Yaskawa INFORM job: SKRZYNIA_5040_90_STOPNI_20BR.JBI

/JOB
//NAME SKRZYNIA_5040_90_STOPNI_20BR
///FOLDERNAME 02-SKRZYNIE_JOBS
//POS
///NPOS 545,545,0,38,0,0
///TOOL 0
///POSTYPE PULSE
///PULSE
C00000=0,-52280,40443,0,6876,0
C00001=82314,-24956,17040,59626,-27382,6248
C00002=93910,-8625,17040,59626,-43355,6248
C00003=98846,-1061,-42166,80308,-57081,-16120
C00004=100452,6057,-48127,85711,-56704,-21322
C00005=95573,33077,-33257,84645,-64023,-26851
C00006=94102,33899,-31937,85246,-63371,-26689
C00007=95573,33077,-33257,84645,-64023,-26851
C00008=94862,31071,-36438,85313,-63677,-27192
C00009=95573,33077,-33257,84645,-64023,-26851
C00010=95263,33142,-33256,84677,-63995,-26850
C00011=95263,33142,-33256,84677,-63995,-26850
C00012=94017,33843,-32133,85187,-63445,-26710
C00013=95263,33142,-33256,84677,-63995,-26850
C00014=94657,31439,-35966,85248,-63701,-27141
C00015=95263,33142,-33256,84677,-63995,-26850
C00016=95260,33144,-33256,84678,-63995,-26850
C00017=95260,33144,-33256,84678,-63995,-26850
C00018=94022,33838,-32141,85183,-63448,-26711
C00019=95260,33144,-33256,84678,-63995,-26850
C00020=94618,31343,-36117,85281,-63684,-27157
C00021=95260,33144,-33256,84678,-63995,-26850
C00022=95258,25631,32269,66559,-75499,-2416
C00023=95258,25631,32269,66559,-75499,-2416
C00024=94181,26497,33533,66410,-74896,-2191
C00025=95658,30184,39035,66708,-78559,-2356
C00026=95217,30377,39331,66881,-79841,-2558
C00027=95258,25631,32269,66559,-75499,-2416
C00028=98811,21047,-15512,99242,-81394,-20987
C00029=98811,21047,-15512,99242,-81394,-20987
C00030=97775,21639,-14693,99563,-80753,-20993
C00031=98811,21047,-15512,99242,-81394,-20987
C00032=98206,18840,-18520,99489,-81124,-21211
C00033=98811,21047,-15512,99242,-81394,-20987
C00034=98765,34858,63506,90961,-74847,-417
C00035=98765,34858,63506,90961,-74847,-417
C00036=97741,35895,65220,90657,-74158,-246
C00037=98765,34858,63506,90961,-74847,-417
C00038=98337,32226,59232,91111,-74633,-884
C00039=98765,34858,63506,90961,-74847,-417
C00040=98728,21792,17445,103800,-78809,-12049
C00041=97232,27021,37502,101932,-75086,-7690
C00042=96358,27701,38514,101868,-74464,-7680
C00043=97232,27021,37502,101932,-75086,-7690
C00044=96733,24820,34282,102049,-74905,-7989
C00045=97232,27021,37502,101932,-75086,-7690
C00046=94428,854,16076,89248,-50738,-4740
C00047=88080,-20128,-3199,80943,-31244,-2335
C00048=48287,-44591,-17414,16172,-14532,25809
C00049=48287,-44591,-17414,16172,-14532,25809
C00050=85348,-13130,13838,41209,-47455,8220
C00051=97395,20012,29210,69700,-74457,-9077
C00052=97055,28839,36684,71776,-79389,-10554
C00053=97055,28839,36684,71776,-79389,-10554
C00054=96058,29646,37897,71666,-78799,-10362
C00055=97055,28839,36684,71776,-79389,-10554
C00056=96570,26659,33451,71832,-78911,-10777
C00057=97055,28839,36684,71776,-79389,-10554
C00058=99123,23256,18377,81563,-78104,3156
C00059=99123,23256,18377,81563,-78104,3156
C00060=98123,23909,19300,81582,-77442,3256
C00061=99123,23256,18377,81563,-78104,3156
C00062=98765,21723,16234,81638,-77830,3017
C00063=99123,23256,18377,81563,-78104,3156
C00064=99222,23346,17795,82202,-78388,4176
C00065=99222,23346,17795,82202,-78388,4176
C00066=98149,24045,18779,82229,-77677,4281
C00067=99222,23346,17795,82202,-78388,4176
C00068=98861,21801,15633,82278,-78114,4033
C00069=99222,23346,17795,82202,-78388,4176
C00070=100468,18781,12295,88713,-76630,3899
C00071=100488,13084,3722,91602,-74275,2573
C00072=99329,-2479,-35949,113241,-72472,-2557
C00073=60067,-64368,-72505,144806,-26050,-19168
C00074=60067,-50244,-32501,110603,-14199,-2207
C00075=63330,-26972,24478,18707,-56801,31483
C00076=95462,-32664,-40336,69376,-39980,4046
C00077=97787,-9790,-26685,81509,-54738,-4408
C00078=99864,21793,7359,80466,-76601,-6182
C00079=99862,21793,7358,80466,-76600,-6182
C00080=98290,21024,6297,80683,-75539,-6194
C00081=97471,21541,7008,80756,-75007,-6115
C00082=98290,21024,6297,80683,-75539,-6194
C00083=97834,19245,3873,80814,-75197,-6333
C00084=98290,21024,6297,80683,-75539,-6194
C00085=98946,26804,31705,85784,-78857,-1423
C00086=98946,26804,31705,85784,-78857,-1423
C00087=98292,27270,32391,85749,-78414,-1361
C00088=98946,26804,31705,85784,-78857,-1423
C00089=98631,25349,29587,85839,-78632,-1590
C00090=98946,26804,31705,85784,-78857,-1423
C00091=94295,-1388,2615,87521,-55608,-1527
C00092=73503,-30722,-22703,70949,-18863,5788
C00093=42754,-66126,12236,-1301,3231,7194
C00094=0,-52280,40443,0,6876,0
C00095=0,-52280,40443,0,6876,0
C00096=48041,-29633,723,44271,-15597,-57965
C00097=51081,-17733,11598,53117,-16128,-61899
C00098=49703,-16390,12674,51759,-15261,-61403
C00099=50366,-16427,12642,52774,-15606,-61824
C00100=49536,-18455,11034,50297,-15435,-60714
C00101=50509,-19000,10610,51503,-15997,-61182
C00102=50873,-17966,11417,52677,-16048,-61710
C00103=49459,-16590,12517,51258,-15158,-61190
C00104=50592,-16429,12648,53120,-15720,-61960
C00105=50873,-17966,11417,52677,-16048,-61710
C00106=50703,-18403,11066,52155,-16024,-61477
C00107=50703,-18403,11066,52155,-16024,-61477
C00108=49026,-16768,12358,50435,-14971,-60844
C00109=50653,-16371,12680,53228,-15754,-62008
C00110=50703,-18403,11066,52155,-16024,-61477
C00111=50704,-18401,11069,52157,-16021,-61478
C00112=50704,-20525,5414,58956,-14779,-64789
C00113=49025,-18889,6668,57745,-13658,-64384
C00114=50799,-18420,7036,60610,-14610,-65581
C00115=50704,-20525,5414,58956,-14779,-64789
C00116=51005,-17995,11387,52847,-16122,-61778
C00117=51005,-17995,11387,52847,-16122,-61778
C00118=49564,-16598,12501,51417,-15218,-61257
C00119=50954,-16306,12737,53719,-15902,-62212
C00120=51005,-17995,11387,52847,-16122,-61778
C00121=51030,-17981,11395,52891,-16138,-61796
C00122=51030,-17981,11395,52891,-16138,-61796
C00123=49401,-16396,12662,51265,-15114,-61201
C00124=50908,-16047,12947,53789,-15850,-62250
C00125=51030,-17981,11395,52891,-16138,-61796
C00126=50945,-18019,11363,52741,-16103,-61737
C00127=50945,-16980,14081,49884,-16761,-60338
C00128=49117,-15186,15539,47848,-15653,-59576
C00129=50939,-14679,15960,50992,-16487,-60881
C00130=50945,-18019,11363,52741,-16103,-61737
C00131=50945,-18019,11363,52741,-16103,-61737
C00132=50945,-18556,9943,54337,-15776,-62517
C00133=48967,-16606,11493,52445,-14510,-61829
C00134=51083,-15952,12027,56053,-15559,-63336
C00135=50945,-18556,9943,54337,-15776,-62517
C00136=50945,-18019,11363,52741,-16103,-61737
C00137=51350,-15183,18375,46705,-17991,-58719
C00138=49319,-13187,20053,44263,-16830,-57796
C00139=51236,-12618,20544,47529,-17647,-59142
C00140=51350,-15183,18375,46705,-17991,-58719
C00141=50028,-23690,-6096,22921,-31075,-54538
C00142=50670,-23735,-6923,24003,-30760,-55076
C00143=48518,-21492,-5254,21861,-29696,-54082
C00144=50138,-21068,-4928,23831,-30039,-55022
C00145=50670,-23735,-6923,24003,-30760,-55076
C00146=49763,-24225,-29961,22080,-30065,-59113
C00147=49763,-24225,-29961,22080,-30065,-59113
C00148=47727,-21550,-27874,20313,-29013,-58119
C00149=49271,-21042,-27466,22016,-29310,-59069
C00150=49763,-24225,-29961,22080,-30065,-59113
C00151=50713,-12366,-58367,41124,-17813,-74400
C00152=50713,-12366,-58367,41124,-17813,-74400
C00153=48934,-9522,-55687,39981,-16902,-73526
C00154=50242,-8975,-55157,41389,-17374,-74448
C00155=50713,-12366,-58367,41124,-17813,-74400
C00156=49763,-25421,-36239,24565,-26935,-60445
C00157=43547,-31626,-19626,5157,-49140,-52118
C00158=40154,-51179,-915,24203,-8234,-36524
C00159=0,-52280,40443,0,6876,0
C00160=0,-52280,40443,0,6876,0
C00161=2117,-50103,-33543,4117,45077,-85249
C00162=-26439,-48928,-33543,4117,-52362,-85249
C00163=-1453,-29933,-32011,46693,-66666,-90474
C00164=24798,-19255,-10490,69050,-85424,-90395
C00165=18386,-22028,-12683,68302,-81515,-89477
///LIMIT ON
C00166=9843,-31743,-57176,61611,-65235,-99401
C00167=-39603,-23393,-71448,91573,-31907,-107123
C00168=-35705,5077,-63140,100511,-35979,-118164
C00169=-33789,12193,-59259,102607,-37482,-119984
C00170=-34998,13124,-58049,103267,-36945,-119997
C00171=-34401,14597,-56112,102586,-37131,-119778
C00172=-34998,13124,-58049,103267,-36945,-119997
C00173=-36388,13885,-57049,104079,-36338,-120048
C00174=-34998,13124,-58049,103267,-36945,-119997
C00175=-34008,-7969,-75285,118537,-50852,-116988
C00176=-26318,8527,-57077,128458,-81874,-108613
///LIMIT OFF
C00177=-23139,-1795,-12064,73373,-53703,-87448
C00178=-27830,-667,-10848,73187,-50621,-86997
C00179=-27373,916,-9115,73207,-50922,-87041
C00180=-27830,-667,-10848,73187,-50621,-86997
C00181=-28901,-207,-10348,73132,-49918,-86888
C00182=-27830,-667,-10848,73187,-50621,-86997
C00183=-37166,8347,13175,41366,-53536,-76331
C00184=-37403,7707,12401,41298,-53388,-76282
C00185=-36830,9273,14303,41455,-53750,-76396
C00186=-37403,7707,12401,41298,-53388,-76282
C00187=-38235,8246,13056,40951,-53040,-76025
C00188=-37403,7707,12401,41298,-53388,-76282
C00189=-30063,5992,18551,55847,-56234,-77619
C00190=-30754,7414,19761,55747,-55713,-77591
C00191=-30376,8670,21285,55817,-55984,-77619
C00192=-30754,7414,19761,55747,-55713,-77591
C00193=-31265,7672,20073,55566,-55435,-77478
C00194=-30085,6037,18588,55845,-56218,-77619
C00195=-25385,-1715,-9470,94765,-53990,-89712
C00196=-25885,-764,-8323,94779,-53645,-89697
C00197=-25564,418,-7032,94741,-53861,-89683
C00198=-25885,-764,-8323,94779,-53645,-89697
C00199=-26741,-428,-7957,94890,-53068,-89741
C00200=-25421,-1648,-9389,94767,-53966,-89710
C00201=-17789,-39335,-40320,90232,-41783,-86178
C00202=-25885,-761,-8324,94780,-53645,-89696
C00203=-25885,-761,-8324,94780,-53645,-89696
C00204=-25612,239,-7230,94748,-53828,-89684
C00205=-25885,-761,-8324,94780,-53645,-89696
C00206=-26712,-436,-7972,94885,-53087,-89742
C00207=-25885,-761,-8324,94780,-53645,-89696
C00208=-26038,-1317,-8919,94796,-53541,-89701
C00209=-18430,-29121,-33898,93348,-44706,-88207
C00210=-3209,-48313,-44409,84985,-37126,-83197
C00211=-3617,-53456,-46461,81793,-37023,-81323
C00212=-28991,-22310,-29554,94749,-46554,-89251
C00213=-30664,-6343,-14094,96248,-45630,-90223
C00214=-30664,-6343,-14094,96248,-45630,-90223
C00215=-30207,-5031,-12762,96238,-45949,-90236
C00216=-30664,-6343,-14094,96248,-45630,-90223
C00217=-31510,-5971,-13720,96406,-45066,-90297
C00218=-29506,-9179,-17232,96085,-46411,-90159
C00219=-30003,-8487,-16482,96169,-46079,-90194
C00220=-30881,-6301,-14053,96286,-45485,-90239
C00221=-30407,-4956,-12684,96275,-45813,-90252
C00222=-30881,-6301,-14053,96286,-45485,-90239
C00223=-31646,-5963,-13712,96429,-44974,-90305
C00224=-29893,-8752,-16772,96152,-46152,-90188
C00225=-30350,-7636,-15544,96220,-45845,-90215
C00226=-30881,-6301,-14053,96286,-45485,-90239
C00227=-30396,-4924,-12652,96275,-45822,-90251
C00228=-30881,-6301,-14053,96286,-45485,-90239
C00229=-31665,-5954,-13703,96434,-44961,-90308
C00230=-29959,-8593,-16598,96162,-46108,-90192
C00231=-26558,-19284,-27675,95285,-48332,-89713
C00232=-5136,-57382,-50746,80999,-31115,-81799
C00233=-5136,-57382,-50746,80999,-31115,-81799
C00234=-22762,-12288,-20025,94001,-55646,-89200
C00235=-24763,-3131,-11201,94769,-54426,-89746
C00236=-26203,-419,-7954,94818,-53430,-89712
C00237=-25939,548,-6896,94784,-53609,-89698
C00238=-26203,-419,-7954,94818,-53430,-89712
C00239=-26818,-174,-7689,94897,-53016,-89744
C00240=-24998,-2701,-10694,94780,-54264,-89743
C00241=-23275,-722,28392,94611,-50650,-77911
C00242=-21733,-16242,25206,75334,-39210,-63099
C00243=0,-52280,40443,0,6876,0
C00244=0,-52280,40443,0,6876,0
C00245=82314,-24956,17040,59626,-27382,6248
C00246=93910,-8625,17040,59626,-43355,6248
C00247=98846,-1061,-42166,80308,-57081,-16120
C00248=100452,6057,-48127,85711,-56704,-21322
C00249=95564,34698,-34234,85516,-63941,-27819
C00250=93687,36612,-31081,84292,-64733,-27467
C00251=93711,36598,-31105,84282,-64744,-27471
C00252=95564,34698,-34234,85516,-63941,-27819
C00253=96930,32282,-32252,82595,-65816,-26305
C00254=93663,32611,-31732,84127,-64318,-26195
C00255=93663,32611,-31732,84127,-64318,-26195
C00256=96930,32282,-32252,82595,-65816,-26305
C00257=96528,-7533,-34932,76119,-53878,-10439
C00258=88377,-34186,-45291,67238,-52212,-2442
C00259=73560,-62084,7826,28695,-34737,3666
C00260=0,-52280,40443,0,6876,0
C00261=0,-52280,40443,0,6876,0
C00262=2117,-50103,-33543,4117,45077,-85249
C00263=-26439,-48928,-33543,4117,-52362,-85249
C00264=-26439,-27355,-33543,41485,-52362,-85249
C00265=-39218,-24492,-41653,51934,-39374,-86964
C00266=-37997,-10433,-19136,70610,-34172,-88069
C00267=-38397,-8978,-17736,70703,-33874,-88109
C00268=-39218,-24492,-41653,51934,-39374,-86964
C00269=-26439,-27355,-33543,41485,-52362,-85249
C00270=1598,-24403,-16502,45671,-72599,-88798
C00271=-11365,-15171,10010,30164,-77975,-82960
C00272=-38112,4197,-14374,43778,-42973,-90436
C00273=-39116,7904,-10019,43942,-43580,-90646
C00274=-38495,8531,-9262,44482,-44499,-91194
C00275=-38112,4197,-14374,43778,-42973,-90436
C00276=-53220,-12364,-8957,19277,-47766,-73858
C00277=-11365,-15171,10010,30164,-77975,-82960
C00278=-16156,-38280,11293,23671,-42998,-42040
C00279=-11365,-47379,10010,30164,3063,-681
C00280=0,-52280,40443,0,6876,0
C00281=0,-36700,24612,-42871,-31823,-33862
C00282=44403,-30110,7154,24155,-23805,-45557
C00283=51347,-17798,16373,37641,-23556,-51399
C00284=51570,-17239,16856,38066,-23574,-51584
C00285=66153,-16343,3873,86567,-32078,-80939
C00286=60867,-15143,12446,70239,-26750,-71065
C00287=40431,-28773,9158,17648,-23273,-42875
C00288=0,-36700,24612,-42871,-31823,-33862
C00289=0,-52280,40443,0,6876,0
C00290=0,-52280,40443,0,6876,0
C00291=73560,-62084,7826,28695,-34737,3666
C00292=88377,-34186,-45291,67238,-52212,-2442
C00293=96528,-7533,-34932,76119,-53878,-10439
C00294=100432,21324,12575,83706,-77956,-7498
C00295=100432,21324,12575,83706,-77956,-7498
C00296=97224,21170,12361,83970,-75786,-7447
C00297=97224,21170,12361,83970,-75786,-7447
C00298=100432,21324,12575,83706,-77956,-7498
C00299=100432,21324,12575,83706,-77956,-7498
C00300=97481,25108,17890,83512,-78432,-7131
C00301=97624,25049,17805,83504,-78528,-7141
C00302=100432,21324,12575,83706,-77956,-7498
C00303=97137,1790,-11103,86179,-63102,-7963
C00304=99183,2264,5333,86781,-62651,-3264
C00305=99868,-33,22146,72719,-59601,5126
C00306=99028,-10516,17309,71061,-60695,4227
C00307=58820,-39124,10926,53325,-41870,3759
C00308=0,-52280,40443,0,6876,0
C00309=37281,-50778,-9546,79570,-75313,-71156
C00310=21038,-23698,-30323,82948,-81132,-85647
C00311=-27256,-5882,-14331,85818,-48304,-85968
C00312=-24751,2890,-4920,85349,-55822,-86178
C00313=-24793,2953,-4845,85351,-55796,-86173
C00314=-27256,-5882,-14331,85818,-48304,-85968
C00315=-21143,-15675,-23596,84785,-52496,-85466
C00316=35274,-15248,-23220,82440,-90817,-86704
C00317=35274,-15248,-23220,82440,-90817,-86704
C00318=-45551,161,-18089,35087,-36064,-73293
C00319=-42435,6767,-10562,40540,-41185,-77662
C00320=-42821,6494,-10882,40094,-40673,-77276
C00321=-45551,161,-18089,35087,-36064,-73293
C00322=-32891,-7184,-22739,69075,-41395,-83248
C00323=-29265,-39765,-39402,58096,-43152,-73226
C00324=-37287,-55159,35520,2191,5667,-2084
C00325=0,-52280,40443,0,6876,0
C00326=0,-36700,24612,-42871,-31823,-33862
C00327=44403,-30110,7154,24155,-23805,-45557
C00328=44403,-30110,7154,24155,-23805,-45557
C00329=42101,-12213,25656,103795,-5192,-78630
C00330=46259,-8171,27719,110365,-8144,-81138
C00331=52601,-3768,32601,101908,-15442,-75329
C00332=54816,-2686,28547,120739,-21736,-87509
C00333=50677,-23266,8367,38735,-22212,-52049
C00334=47073,-34549,9488,27883,-30316,-51458
C00335=0,-52280,40443,0,6876,0
C00336=0,-52280,40443,0,6876,0
C00337=73560,-62084,7826,28695,-34737,3666
C00338=96983,-27116,-23481,78724,-62297,-1998
C00339=100467,-7393,-15195,81625,-60158,-6002
C00340=99336,18440,8642,84276,-74234,-7647
C00341=99336,18440,8642,84276,-74234,-7647
C00342=97735,24994,14595,85350,-78994,-5109
C00343=97744,25074,13580,86004,-79195,-4385
C00344=99336,18440,8642,84276,-74234,-7647
C00345=99336,18440,8642,84276,-74234,-7647
C00346=97891,23737,8261,88167,-79183,-2386
C00347=97851,23541,8142,88101,-79081,-2507
C00348=99336,18440,8642,84276,-74234,-7647
C00349=89817,-17341,-38408,97132,-45323,-12250
C00350=100347,-21961,-42251,93939,-52125,-11121
C00351=60204,-59872,-73451,117647,-17639,-18840
C00352=37721,-67612,11381,1325,-438,7850
C00353=-37287,-55159,35520,2191,5667,-2084
C00354=-40042,-68802,-18337,47708,-19461,-45384
C00355=-28646,-23138,-32952,89786,-42552,-85395
C00356=-38882,-16596,-17625,44304,-41043,-72768
C00357=-42680,-6319,-12818,46127,-36112,-73823
C00358=-37459,704,-5408,52536,-43357,-78192
C00359=-32778,4349,-7465,59128,-48375,-83352
C00360=-42680,-6319,-12818,46127,-36112,-73823
C00361=-38882,-16596,-17625,44304,-41043,-72768
C00362=-28646,-23138,-32952,89786,-42552,-85395
C00363=-29905,-15291,-26411,91102,-43435,-86304
C00364=-25469,1350,-9790,89991,-54827,-86555
C00365=-24242,3379,-7505,89554,-57286,-86471
C00366=-29905,-15291,-26411,91102,-43435,-86304
C00367=-40042,-68802,-18337,47708,-19461,-45384
C00368=-37287,-55159,35520,2191,5667,-2084
C00369=0,-52280,40443,0,6876,0
C00370=37164,-60659,6466,13301,-5027,-19773
C00371=45362,-39990,2831,27538,-17767,-40935
C00372=57189,-26834,-7130,38780,-31731,-51561
C00373=63456,-14144,8594,45591,-40850,-50620
C00374=63298,-23815,-40708,66066,-30898,-63274
C00375=57189,-26834,-7130,38780,-31731,-51561
C00376=41180,-61187,4729,17280,-8498,-23442
C00377=0,-52280,40443,0,6876,0
C00378=0,-52280,40443,0,6876,0
C00379=37721,-67612,11381,1325,-438,7850
C00380=43180,-50572,-20637,6552,-29302,38834
C00381=79425,-37128,-15462,51820,-35721,18807
C00382=93702,-21743,-5664,65079,-41536,12324
C00383=94876,-11469,-23586,124528,-59237,-5423
C00384=92578,22421,15997,116595,-76671,1441
C00385=90287,21612,15190,116916,-75301,1087
C00386=91032,29854,33392,114957,-76206,4791
C00387=92578,22421,15997,116595,-76671,1441
C00388=94876,-11469,-23586,124528,-59237,-5423
C00389=93702,-22946,-9336,66730,-40927,11282
C00390=92743,-25622,-14104,67700,-39874,10604
C00391=95618,-29588,-12765,65168,-50072,21743
C00392=-36913,-32963,-979,75363,-26772,-58744
C00393=-42264,1508,8544,35869,-47237,-69477
C00394=-43183,4597,12058,35318,-46938,-69128
C00395=-43183,5775,16318,34276,-48598,-68388
C00396=-42264,1508,8544,35869,-47237,-69477
C00397=56258,-38103,3288,28818,-33580,-23051
C00398=41438,-37635,17580,13151,-29920,-38779
C00399=54964,-26842,8528,44141,-23181,-52038
C00400=50761,-21373,7883,46957,-18149,-54038
C00401=65214,-17346,-4869,103105,-32325,-89305
C00402=65312,-6152,27526,81270,-31139,-77237
C00403=56762,-20631,11812,69834,-24329,-69917
C00404=46096,-45842,-2681,20981,-19497,-36310
C00405=41180,-61187,4729,17280,-8498,-23442
C00406=0,-52280,40443,0,6876,0
C00407=0,-52280,40443,0,6876,0
C00408=37721,-67612,11381,1325,-438,7850
C00409=43180,-50572,-20637,6552,-29302,38834
C00410=79425,-37128,-15462,51820,-35721,18807
C00411=92377,-33385,-41303,83059,-36844,1354
C00412=97441,-6012,-18634,86114,-58345,-2339
C00413=98864,-2001,-14672,90389,-62789,-3799
C00414=98767,21176,13691,87588,-77304,-2577
C00415=98123,23617,17097,87345,-78645,-2335
C00416=97979,23711,17231,87352,-78549,-2326
C00417=98864,-2001,-14672,90389,-62789,-3799
C00418=100472,-329,-13432,98539,-67097,-6304
C00419=92822,-26306,-37175,103295,-43881,-7703
C00420=68601,-52593,-52127,95725,-25602,-3235
C00421=80632,-38079,-20908,64053,-45216,12949
C00422=43180,-50572,-20637,6552,-29302,38834
C00423=37721,-67612,11381,1325,-438,7850
C00424=0,-52280,40443,0,6876,0
C00425=0,-52280,40443,0,6876,0
C00426=0,-52280,40443,0,-39412,36675
C00427=-54026,-30203,28811,-7745,-28969,-5087
C00428=-30389,-9386,-5824,79667,-43789,-73484
C00429=-32979,-3325,255,79720,-41988,-73575
C00430=-25304,6223,10893,81656,-55729,-74481
C00431=-23842,8927,14147,81883,-58875,-74544
C00432=-30389,-9386,-5824,79667,-43789,-73484
C00433=-32145,-6440,-2937,79673,-42575,-73527
C00434=-25014,6414,11121,81706,-56254,-74506
C00435=-23603,11547,23533,79434,-59735,-72187
C00436=-32145,-5050,2357,77009,-42992,-71800
C00437=-35251,-18143,20376,53513,-41117,-59413
C00438=-9534,-43450,13514,26959,-29486,-38723
C00439=-22834,-59963,22946,6692,-2150,-9612
C00440=0,-52280,40443,0,6876,0
C00441=23708,-46776,23536,16027,-4787,-19738
C00442=50917,-40459,4132,34421,-18173,-42391
C00443=51059,-36587,4608,36647,-19418,-45358
C00444=50113,-22729,10834,36393,-23396,-50963
C00445=62046,-17757,4067,79440,-27252,-76630
C00446=63804,-15651,7512,80030,-29507,-77065
C00447=50113,-22729,10834,36393,-23396,-50963
C00448=31287,-69981,-10850,7253,-6843,-20996
C00449=19644,-57271,30737,863,5243,-2499
C00450=0,-52280,40443,0,6876,0
C00451=0,-52280,40443,0,6876,0
C00452=37721,-67612,11381,1325,-438,7850
C00453=43180,-50572,-20637,6552,-29302,38834
C00454=79425,-37128,-15462,51820,-35721,18807
C00455=92377,-33385,-41303,83059,-36844,1354
C00456=97441,-6012,-18634,86114,-58345,-2339
C00457=98442,-3149,-15680,86092,-59018,-2413
C00458=96855,-5742,-18360,86176,-57949,-2343
C00459=99185,22470,15697,83135,-77937,-1734
C00460=97717,21807,14770,83256,-76932,-1762
C00461=97717,21807,14770,83256,-76932,-1762
C00462=99185,24652,26607,82087,-78431,1026
C00463=99185,22470,15697,83135,-77937,-1734
C00464=97852,24994,19264,82957,-78889,-1504
C00465=97683,25109,19429,82963,-78778,-1488
C00466=99870,24121,23963,82328,-78767,341
C00467=100471,12680,2182,89317,-73847,-3746
C00468=93923,-8883,-21959,92925,-54783,-4609
C00469=92822,-26306,-37175,103295,-43881,-7703
C00470=68601,-52593,-52127,95725,-25602,-3235
C00471=80632,-38079,-20908,64053,-45216,12949
C00472=43180,-50572,-20637,6552,-29302,38834
C00473=37721,-67612,11381,1325,-438,7850
C00474=0,-52280,40443,0,6876,0
C00475=0,-52280,40443,0,6876,0
C00476=0,-52280,40443,0,-39412,36675
C00477=-54026,-30203,28811,-7745,-28969,-5087
C00478=-81492,-18979,22896,-11682,-23662,-26316
C00479=-32145,-2720,10458,73217,-43826,-69319
C00480=-32145,-2720,10458,73217,-43826,-69319
C00481=-25800,12961,35355,74076,-56913,-68018
C00482=-23961,12723,28512,77913,-59573,-70804
C00483=-32145,-2720,10458,73217,-43826,-69319
C00484=-34274,-9754,-24316,117159,-46217,-86271
C00485=-34274,-9754,-24316,117159,-46217,-86271
C00486=-29822,-1437,-15851,112752,-53901,-84078
C00487=-28945,-336,-14662,112011,-55335,-83695
C00488=-34274,-9754,-24316,117159,-46217,-86271
C00489=-34422,-9999,20796,72411,-42519,-66994
C00490=-35251,-18143,20376,53513,-41117,-59413
C00491=-9534,-43450,13514,26959,-29486,-38723
C00492=-22834,-59963,22946,6692,-2150,-9612
C00493=0,-52280,40443,0,6876,0
C00494=44101,-76445,-48847,15697,-17168,-40457
C00495=49121,-28282,-35458,21895,-29219,-59001
C00496=50484,-13386,-55713,36158,-19724,-71897
C00497=55938,-10187,-55661,55618,-22248,-82832
C00498=57381,15206,-57369,78100,-21009,-89969
C00499=50484,-13386,-55713,36158,-19724,-71897
C00500=49763,-25421,-36239,24565,-26935,-60445
C00501=50529,-22709,-3778,22940,-31995,-54502
C00502=45389,-28224,4312,35967,-15579,-54278
C00503=40154,-51179,-915,24203,-8234,-36524
C00504=0,-52280,40443,0,6876,0
C00505=0,-52280,40443,0,6876,0
C00506=37721,-67612,11381,1325,-438,7850
C00507=43181,-50571,-20637,6551,-29300,38834
C00508=92325,-23846,-7228,63960,-40898,12897
C00509=85232,-2754,25377,50981,-49542,17626
C00510=95618,10017,30418,66150,-65403,10402
C00511=98328,26728,37723,75385,-78922,5377
C00512=97988,24882,21615,85608,-78767,-653
C00513=97988,24882,21615,85608,-78767,-653
C00514=97883,29022,44703,72741,-79810,7156
C00515=99525,21729,17159,85870,-76787,-954
C00516=97991,25479,22462,85564,-79108,-597
C00517=97991,25479,22462,85564,-79108,-597
C00518=99525,21729,17159,85870,-76787,-954
C00519=85644,-12525,-7527,79034,-40769,5189
C00520=97513,-10257,11960,71433,-51152,11355
C00521=72477,-33752,-3372,52810,-39669,19964
C00522=0,-52278,40443,0,6872,5
C00523=0,-52278,40443,31822,-65283,-46097
C00524=-7820,3000,44222,77356,-66876,-70486
C00525=-24244,23423,72059,64993,-61079,-67138
C00526=-27261,30732,84230,62108,-60720,-65392
C00527=-22394,37028,87531,68934,-68535,-64461
C00528=-24244,23423,72059,64993,-61079,-67138
C00529=3014,-20441,-7349,104591,-68614,-79454
C00530=6322,-14118,13197,96169,-69167,-72790
C00531=14133,-16757,18528,88010,-59455,-67296
C00532=-10261,-46634,14475,36899,-22136,-31570
C00533=-22834,-59963,22946,6692,-2150,-9612
C00534=0,-52280,40443,0,6876,0
C00535=23708,-46776,23536,16027,-4787,-19738
C00536=50917,-40459,4132,34421,-18173,-42391
C00537=49876,-21948,7530,68838,-10324,-59148
C00538=46721,-18942,9765,68167,-8197,-59205
C00539=59102,-15651,-1637,118714,-27356,-88041
C00540=59185,-13834,7185,105143,-23914,-78054
C00541=45927,-22803,4403,78462,-8511,-64553
C00542=62498,-35400,-2607,72048,-19281,-59202
C00543=31287,-69981,-10850,7253,-6843,-20996
C00544=0,-52280,40443,0,6876,0
BC00000=487510
BC00001=445130
BC00002=445130
BC00003=445130
BC00004=445130
BC00005=468227
BC00006=468227
BC00007=468227
BC00008=468227
BC00009=468227
BC00010=514421
BC00011=514421
BC00012=514421
BC00013=514421
BC00014=514421
BC00015=514421
BC00016=560588
BC00017=560588
BC00018=560588
BC00019=560588
BC00020=560588
BC00021=560588
BC00022=536404
BC00023=536404
BC00024=536404
BC00025=536404
BC00026=536404
BC00027=536404
BC00028=582458
BC00029=582458
BC00030=582458
BC00031=582458
BC00032=582458
BC00033=582458
BC00034=581206
BC00035=581206
BC00036=581206
BC00037=581206
BC00038=581206
BC00039=581206
BC00040=626960
BC00041=626960
BC00042=626960
BC00043=626960
BC00044=626960
BC00045=626960
BC00046=604255
BC00047=604255
BC00048=604255
BC00049=699121
BC00050=714117
BC00051=772491
BC00052=770398
BC00053=770398
BC00054=770398
BC00055=770398
BC00056=770398
BC00057=770398
BC00058=820815
BC00059=820815
BC00060=820815
BC00061=820815
BC00062=820815
BC00063=820815
BC00064=866263
BC00065=866263
BC00066=866260
BC00067=866263
BC00068=866263
BC00069=866263
BC00070=868226
BC00071=868803
BC00072=869038
BC00073=872244
BC00074=872244
BC00075=914118
BC00076=976590
BC00077=976703
BC00078=976734
BC00079=964492
BC00080=964492
BC00081=964492
BC00082=964492
BC00083=964492
BC00084=964492
BC00085=963886
BC00086=963886
BC00087=963886
BC00088=963886
BC00089=963886
BC00090=963886
BC00091=945942
BC00092=953277
BC00093=857759
BC00094=811793
BC00095=811793
BC00096=953382
BC00097=953382
BC00098=953382
BC00099=953383
BC00100=953382
BC00101=888056
BC00102=888056
BC00103=888056
BC00104=888056
BC00105=888056
BC00106=830714
BC00107=830714
BC00108=830714
BC00109=830714
BC00110=830714
BC00111=764829
BC00112=764829
BC00113=764829
BC00114=764829
BC00115=764829
BC00116=707174
BC00117=707174
BC00118=707174
BC00119=707174
BC00120=707174
BC00121=642071
BC00122=642071
BC00123=642071
BC00124=642071
BC00125=642071
BC00126=584746
BC00127=584746
BC00128=584746
BC00129=584746
BC00130=584746
BC00131=519232
BC00132=519232
BC00133=519232
BC00134=519232
BC00135=519232
BC00136=461813
BC00137=461813
BC00138=461813
BC00139=461813
BC00140=461813
BC00141=459544
BC00142=459544
BC00143=459544
BC00144=459544
BC00145=459544
BC00146=459544
BC00147=459544
BC00148=459544
BC00149=459544
BC00150=459544
BC00151=459544
BC00152=459544
BC00153=459544
BC00154=459544
BC00155=459544
BC00156=459544
BC00157=462325
BC00158=533216
BC00159=533216
BC00160=492150
BC00161=423885
BC00162=423885
BC00163=519103
BC00164=542802
BC00165=634915
BC00166=493160
BC00167=493160
BC00168=517936
BC00169=517447
BC00170=516208
BC00171=516208
BC00172=516208
BC00173=516208
BC00174=516208
BC00175=525487
BC00176=485388
BC00177=500803
BC00178=500803
BC00179=500803
BC00180=500803
BC00181=500803
BC00182=500803
BC00183=585253
BC00184=585253
BC00185=585253
BC00186=585253
BC00187=585253
BC00188=585253
BC00189=600589
BC00190=600589
BC00191=600589
BC00192=600589
BC00193=600589
BC00194=600589
BC00195=646713
BC00196=646713
BC00197=646713
BC00198=646713
BC00199=646713
BC00200=646713
BC00201=659006
BC00202=692822
BC00203=692822
BC00204=692822
BC00205=692822
BC00206=692822
BC00207=692822
BC00208=669701
BC00209=669701
BC00210=669701
BC00211=791136
BC00212=762000
BC00213=762000
BC00214=762000
BC00215=762000
BC00216=762000
BC00217=762000
BC00218=762000
BC00219=831025
BC00220=831025
BC00221=831025
BC00222=831025
BC00223=831025
BC00224=831025
BC00225=877128
BC00226=877128
BC00227=877128
BC00228=877128
BC00229=877128
BC00230=877128
BC00231=854090
BC00232=854090
BC00233=990684
BC00234=992363
BC00235=992364
BC00236=992364
BC00237=992364
BC00238=992364
BC00239=992364
BC00240=992364
BC00241=941750
BC00242=932032
BC00243=834170
BC00244=445130
BC00245=445130
BC00246=445130
BC00247=445130
BC00248=445130
BC00249=475938
BC00250=475938
BC00251=468314
BC00252=475938
BC00253=515329
BC00254=515329
BC00255=507641
BC00256=515329
BC00257=542207
BC00258=542207
BC00259=542207
BC00260=542207
BC00261=492150
BC00262=423885
BC00263=423885
BC00264=423885
BC00265=423885
BC00266=406365
BC00267=406365
BC00268=423885
BC00269=423885
BC00270=423885
BC00271=423885
BC00272=507950
BC00273=507950
BC00274=500226
BC00275=507950
BC00276=493160
BC00277=493160
BC00278=493160
BC00279=493160
BC00280=493160
BC00281=582810
BC00282=655182
BC00283=712102
BC00284=712780
BC00285=712780
BC00286=769565
BC00287=773753
BC00288=582810
BC00289=493160
BC00290=542207
BC00291=542207
BC00292=542207
BC00293=590944
BC00294=543764
BC00295=459277
BC00296=459277
BC00297=451665
BC00298=459277
BC00299=520748
BC00300=520748
BC00301=528468
BC00302=520748
BC00303=524597
BC00304=604006
BC00305=584417
BC00306=584417
BC00307=584417
BC00308=584417
BC00309=542360
BC00310=521200
BC00311=474976
BC00312=474976
BC00313=482600
BC00314=474976
BC00315=474976
BC00316=474976
BC00317=630364
BC00318=628593
BC00319=624867
BC00320=617183
BC00321=631527
BC00322=617183
BC00323=617427
BC00324=620193
BC00325=620193
BC00326=812803
BC00327=887783
BC00328=927066
BC00329=893694
BC00330=914884
BC00331=914884
BC00332=942497
BC00333=962387
BC00334=853059
BC00335=542207
BC00336=542207
BC00337=542207
BC00338=541760
BC00339=590944
BC00340=571989
BC00341=566860
BC00342=566868
BC00343=574636
BC00344=566860
BC00345=635958
BC00346=635958
BC00347=643642
BC00348=635958
BC00349=635118
BC00350=635118
BC00351=656468
BC00352=665809
BC00353=620193
BC00354=620193
BC00355=635598
BC00356=635598
BC00357=635598
BC00358=635598
BC00359=635598
BC00360=635598
BC00361=635598
BC00362=635598
BC00363=658627
BC00364=658627
BC00365=666320
BC00366=658627
BC00367=620193
BC00368=620193
BC00369=620193
BC00370=561542
BC00371=498768
BC00372=452071
BC00373=452071
BC00374=452075
BC00375=452071
BC00376=524165
BC00377=524165
BC00378=733103
BC00379=733103
BC00380=733103
BC00381=615417
BC00382=615411
BC00383=615411
BC00384=615411
BC00385=615411
BC00386=615411
BC00387=615411
BC00388=615411
BC00389=615411
BC00390=615417
BC00391=615413
BC00392=696009
BC00393=735643
BC00394=735643
BC00395=739967
BC00396=735643
BC00397=617218
BC00398=582869
BC00399=580754
BC00400=589556
BC00401=589556
BC00402=626883
BC00403=634257
BC00404=536572
BC00405=561088
BC00406=547800
BC00407=733103
BC00408=733103
BC00409=733103
BC00410=733103
BC00411=733103
BC00412=733103
BC00413=740531
BC00414=740531
BC00415=740531
BC00416=748211
BC00417=740531
BC00418=750469
BC00419=750469
BC00420=750469
BC00421=783373
BC00422=795297
BC00423=733103
BC00424=733103
BC00425=672709
BC00426=672709
BC00427=762701
BC00428=743900
BC00429=736524
BC00430=736351
BC00431=743900
BC00432=743900
BC00433=759331
BC00434=759331
BC00435=759331
BC00436=759331
BC00437=750104
BC00438=672725
BC00439=672725
BC00440=672725
BC00441=766882
BC00442=791101
BC00443=802867
BC00444=836517
BC00445=836517
BC00446=895034
BC00447=836517
BC00448=618402
BC00449=618402
BC00450=618402
BC00451=733103
BC00452=733103
BC00453=733103
BC00454=733103
BC00455=733103
BC00456=733103
BC00457=815683
BC00458=817504
BC00459=817504
BC00460=817504
BC00461=825298
BC00462=817504
BC00463=863642
BC00464=863642
BC00465=871437
BC00466=863642
BC00467=817424
BC00468=817332
BC00469=750469
BC00470=750469
BC00471=783373
BC00472=795297
BC00473=733103
BC00474=733103
BC00475=672709
BC00476=672709
BC00477=762701
BC00478=791880
BC00479=819491
BC00480=819491
BC00481=817331
BC00482=817331
BC00483=817326
BC00484=863478
BC00485=863478
BC00486=863478
BC00487=871062
BC00488=863478
BC00489=774095
BC00490=750104
BC00491=672725
BC00492=672725
BC00493=672725
BC00494=528256
BC00495=459544
BC00496=459544
BC00497=459544
BC00498=459547
BC00499=459544
BC00500=459544
BC00501=459544
BC00502=459540
BC00503=533216
BC00504=533216
BC00505=733103
BC00506=733103
BC00507=945037
BC00508=938671
BC00509=928072
BC00510=935112
BC00511=947035
BC00512=947035
BC00513=954731
BC00514=947035
BC00515=970062
BC00516=970062
BC00517=977728
BC00518=970062
BC00519=975033
BC00520=955597
BC00521=952322
BC00522=852584
BC00523=921533
BC00524=958534
BC00525=946591
BC00526=946591
BC00527=946592
BC00528=954904
BC00529=963295
BC00530=934184
BC00531=908449
BC00532=754884
BC00533=672725
BC00534=672725
BC00535=562340
BC00536=452362
BC00537=452362
BC00538=452362
BC00539=452362
BC00540=513216
BC00541=512110
BC00542=512008
BC00543=742282
BC00544=742282
///POSTYPE BASE
///RECTAN
///RCONF 1,0,0,0,0,0,0,0,0,0,0,0,0,0,0,0,0,0,0,0,0,0,0,0
P00006=-0.064,-0.849,9.145,0.0000,0.0000,0.0000
///RCONF 0,0,0,0,0,0,0,0,0,0,0,0,0,0,0,0,0,0,0,0,0,0,0,0
P00058=0.000,0.000,3.000,0.0000,0.0000,0.0000
///RCONF 1,0,0,0,0,0,0,0,0,0,0,0,0,0,0,0,0,0,0,0,0,0,0,0
P00300=-0.036,-1.505,2.318,0.0000,0.0000,0.0000
///RCONF 0,0,0,0,0,0,0,0,0,0,0,0,0,0,0,0,0,0,0,0,0,0,0,0
P00301=0.005,-4.708,-4.628,0.0000,0.0000,0.0000
P00302=0.052,-2.937,-4.426,0.0000,0.0000,0.0000
P00303=-0.004,-1.437,-4.584,0.0000,0.0000,0.0000
P00304=0.028,-1.666,-4.234,0.0000,0.0000,0.0000
P00305=-0.003,-1.920,-3.501,0.0000,0.0000,0.0000
P00306=0.015,-2.252,-3.054,0.0000,0.0000,0.0000
P00307=0.019,-2.151,-5.077,0.0000,0.0000,0.0000
P00308=-0.003,-2.092,-4.888,0.0000,0.0000,0.0000
P00309=-0.040,-2.205,-4.992,0.0000,0.0000,0.0000
P00310=-0.006,-2.490,-5.925,0.0000,0.0000,0.0000
P00311=-0.007,-2.079,-5.307,0.0000,0.0000,0.0000
P00350=11.519,-0.008,1.149,0.0000,0.0000,0.0000
P00351=13.563,-0.027,-0.653,0.0000,0.0000,0.0000
P00352=13.252,-0.027,-0.827,0.0000,0.0000,0.0000
P00353=10.971,-0.082,0.776,0.0000,0.0000,0.0000
P00354=-0.024,2.508,-1.824,0.0000,0.0000,0.0000
P00355=-0.001,2.528,-1.131,0.0000,0.0000,0.0000
P00356=-0.034,2.921,-0.262,0.0000,0.0000,0.0000
P00357=0.003,3.386,-0.091,0.0000,0.0000,0.0000
P00358=0.014,3.037,-0.020,0.0000,0.0000,0.0000
P00359=-0.005,2.731,0.912,0.0000,0.0000,0.0000
P00360=-0.011,3.412,0.438,0.0000,0.0000,0.0000
P00361=0.018,3.050,1.253,0.0000,0.0000,0.0000
P00400=5.920,-3.503,-0.024,0.0000,0.0000,0.0000
P00401=3.430,-0.021,1.131,0.0000,0.0000,0.0000
P00402=-0.253,1.107,3.062,0.0000,0.0000,0.0000
P00403=-3.666,-0.015,5.328,0.0000,0.0000,0.0000
///RCONF 1,0,0,0,0,0,0,0,0,0,0,0,0,0,0,0,0,0,0,0,0,0,0,0
P00404=0.029,4.189,-1.030,0.0000,0.0000,0.0000
///RCONF 0,0,0,0,0,0,0,0,0,0,0,0,0,0,0,0,0,0,0,0,0,0,0,0
P00405=2.420,0.007,1.427,0.0000,0.0000,0.0000
P00406=3.513,-0.022,0.429,0.0000,0.0000,0.0000
///RCONF 1,0,0,0,1,0,0,0,0,0,0,0,0,0,0,0,0,0,0,0,0,0,0,0
P00407=-0.029,2.348,-1.469,0.0000,0.0000,0.0000
P00408=0.010,1.346,-1.479,0.0000,0.0000,0.0000
///RCONF 1,0,0,0,0,0,0,0,0,0,0,0,0,0,0,0,0,0,0,0,0,0,0,0
P00409=-0.026,2.090,-1.483,0.0000,0.0000,0.0000
P00410=0.001,4.491,-0.583,0.0000,0.0000,0.0000
///RCONF 1,0,0,0,1,0,0,0,0,0,0,0,0,0,0,0,0,0,0,0,0,0,0,0
P00411=-0.015,3.627,0.872,0.0000,0.0000,0.0000
//INST
///DATE 2024/05/16 20:17
///ATTR SC,RW
///GROUP1 RB1,BS1
NOP
CALL JOB:MOVE_INTO_TUNNEL
MOVJ C00000 BC00000 VJ=10.00
MOVJ C00001 BC00001 VJ=30.00
MOVJ C00002 BC00002 VJ=30.00
MOVL C00003 BC00003 V=500.0
MOVJ C00004 BC00004 VJ=30.00
'------------------------
'W65.3
'------------------------
MOVL C00005 BC00005 V=333.3 PL=0
REFP 3 C00006 BC00006
CALL JOB:SEARCH-R1
SET P0300 P0006
SFTON P0300
MOVL C00007 BC00007 V=333.3 PL=0
REFP 3 C00008 BC00008
CALL JOB:SEARCH-R1
SET P0300 P0006
SFTON P0300
MOVL C00009 BC00009 V=333.3 PL=0
SFTOF
'------------------------
'W65.5
'------------------------
MOVL C00010 BC00010 V=500.0
MOVL C00011 BC00011 V=333.3 PL=0
REFP 3 C00012 BC00012
CALL JOB:SEARCH-R1
SET P0301 P0006
SFTON P0301
MOVL C00013 BC00013 V=333.3 PL=0
REFP 3 C00014 BC00014
CALL JOB:SEARCH-R1
SET P0301 P0006
SFTON P0301
MOVL C00015 BC00015 V=333.3 PL=0
SFTOF
'------------------------
'W65.7
'------------------------
MOVL C00016 BC00016 V=500.0
MOVL C00017 BC00017 V=333.3 PL=0
REFP 3 C00018 BC00018
CALL JOB:SEARCH-R1
SET P0302 P0006
SFTON P0302
MOVL C00019 BC00019 V=333.3 PL=0
REFP 3 C00020 BC00020
CALL JOB:SEARCH-R1
SET P0302 P0006
SFTON P0302
MOVL C00021 BC00021 V=500.0 PL=0
SFTOF
'------------------------
'W65.10
'------------------------
MOVL C00022 BC00022 V=500.0
MOVL C00023 BC00023 V=333.3 PL=0
REFP 3 C00024 BC00024
CALL JOB:SEARCH-R1
SET P0303 P0006
SFTON P0303
MOVL C00025 BC00025 V=333.3 PL=0
REFP 3 C00026 BC00026
CALL JOB:SEARCH-R1
SET P0303 P0006
SFTON P0303
MOVL C00027 BC00027 V=333.3 PL=0
SFTOF
'------------------------
'W65.12
'------------------------
MOVL C00028 BC00028 V=500.0
MOVL C00029 BC00029 V=333.3 PL=0
REFP 3 C00030 BC00030
CALL JOB:SEARCH-R1
SET P0304 P0006
SFTON P0304
MOVL C00031 BC00031 V=333.3 PL=0
REFP 3 C00032 BC00032
CALL JOB:SEARCH-R1
SET P0304 P0006
SFTON P0304
MOVL C00033 BC00033 V=333.3 PL=0
SFTOF
'------------------------
'W65.15
'------------------------
MOVL C00034 BC00034 V=500.0
MOVL C00035 BC00035 V=333.3 PL=0
REFP 3 C00036 BC00036
CALL JOB:SEARCH-R1
SET P0305 P0006
SFTON P0305
MOVL C00037 BC00037 V=333.3 PL=0
REFP 3 C00038 BC00038
CALL JOB:SEARCH-R1
SET P0305 P0006
SFTON P0305
MOVL C00039 BC00039 V=333.3 PL=0
SFTOF
'------------------------
'W65.17
'------------------------
MOVL C00040 BC00040 V=500.0
MOVL C00041 BC00041 V=166.7 PL=0
REFP 3 C00042 BC00042
CALL JOB:SEARCH-R1
SET P0306 P0006
SFTON P0306
MOVL C00043 BC00043 V=333.3 PL=0
REFP 3 C00044 BC00044
CALL JOB:SEARCH-R1
SET P0306 P0006
SFTON P0306
MOVL C00045 BC00045 V=500.0 PL=0
SFTOF
MOVL C00046 BC00046 V=500.0
MOVL C00047 BC00047 V=500.0
MOVL C00048 BC00048 V=500.0
MOVJ C00049 BC00049 VJ=30.00
MOVL C00050 BC00050 V=500.0
MOVL C00051 BC00051 V=500.0
'------------------------
'W65.20
'------------------------
MOVL C00052 BC00052 V=500.0
MOVL C00053 BC00053 V=333.3 PL=0
REFP 3 C00054 BC00054
CALL JOB:SEARCH-R1
SET P0307 P0006
SFTON P0307
MOVL C00055 BC00055 V=333.3 PL=0
REFP 3 C00056 BC00056
CALL JOB:SEARCH-R1
SET P0307 P0006
SFTON P0307
MOVL C00057 BC00057 V=500.0 PL=0
SFTOF
'------------------------
'W65.23
'------------------------
MOVL C00058 BC00058 V=500.0
MOVL C00059 BC00059 V=333.3 PL=0
REFP 3 C00060 BC00060
CALL JOB:SEARCH-R1
SET P0308 P0006
SFTON P0308
MOVL C00061 BC00061 V=333.3 PL=0
REFP 3 C00062 BC00062
CALL JOB:SEARCH-R1
SET P0308 P0006
SFTON P0308
MOVL C00063 BC00063 V=500.0 PL=0
SFTOF
'------------------------
'W65.25
'------------------------
MOVL C00064 BC00064 V=500.0
MOVL C00065 BC00065 V=333.3 PL=0
REFP 3 C00066 BC00066
CALL JOB:SEARCH-R1
SET P0309 P0006
SFTON P0309
MOVL C00067 BC00067 V=333.3 PL=0
REFP 3 C00068 BC00068
CALL JOB:SEARCH-R1
SET P0309 P0006
SFTON P0309
MOVL C00069 BC00069 V=500.0 PL=0
SFTOF
MOVL C00070 BC00070 V=500.0
MOVL C00071 BC00071 V=500.0
MOVL C00072 BC00072 V=500.0
MOVL C00073 BC00073 V=500.0
MOVL C00074 BC00074 V=500.0
MOVL C00075 BC00075 V=250.0
MOVL C00076 BC00076 V=500.0
MOVL C00077 BC00077 V=500.0
MOVL C00078 BC00078 V=83.3
'------------------------
'W65.28
'------------------------
MOVL C00079 BC00079 V=500.0
MOVL C00080 BC00080 V=333.3 PL=0
REFP 3 C00081 BC00081
CALL JOB:SEARCH-R1
SET P0310 P0006
SFTON P0310
MOVL C00082 BC00082 V=333.3 PL=0
REFP 3 C00083 BC00083
CALL JOB:SEARCH-R1
SET P0310 P0006
SFTON P0310
MOVL C00084 BC00084 V=333.3 PL=0
SFTOF
'------------------------
'W65.30
'------------------------
MOVL C00085 BC00085 V=500.0
MOVL C00086 BC00086 V=333.3 PL=0
REFP 3 C00087 BC00087
CALL JOB:SEARCH-R1
SET P0311 P0006
SFTON P0311
MOVL C00088 BC00088 V=333.3 PL=0
REFP 3 C00089 BC00089
CALL JOB:SEARCH-R1
SET P0311 P0006
SFTON P0311
MOVL C00090 BC00090 V=333.3 PL=0
SFTOF
MOVL C00091 BC00091 V=500.0
MOVL C00092 BC00092 V=500.0
MOVJ C00093 BC00093 VJ=30.00
MOVJ C00094 BC00094 VJ=30.00
MOVJ C00095 BC00095 VJ=30.00
MOVJ C00096 BC00096 VJ=30.00
'------------------------
'W251A
'------------------------
MOVL C00097 BC00097 V=333.3 PL=0
REFP 3 C00098 BC00098
CALL JOB:SEARCH-R1
IMOV P0058 V=16.7
SET P0350 P0006
SFTON P0350
REFP 3 C00099 BC00099
CALL JOB:SEARCH-R1
SET P0350 P0006
SFTON P0350
MOVL C00100 BC00100 V=500.0 PL=0
SFTOF
'------------------------
'W254A P
'------------------------
MOVJ C00101 BC00101 VJ=30.00
MOVL C00102 BC00102 V=333.3 PL=0
REFP 3 C00103 BC00103
CALL JOB:SEARCH-R1
IMOV P0058 V=16.7
SET P0351 P0006
SFTON P0351
REFP 3 C00104 BC00104
CALL JOB:SEARCH-R1
SET P0351 P0006
SFTON P0351
MOVL C00105 BC00105 V=500.0 PL=0
SFTOF
'------------------------
'W254A L
'------------------------
MOVJ C00106 BC00106 VJ=30.00
MOVL C00107 BC00107 V=333.3 PL=0
REFP 3 C00108 BC00108
CALL JOB:SEARCH-R1
IMOV P0058 V=16.7
SET P0352 P0006
SFTON P0352
REFP 3 C00109 BC00109
CALL JOB:SEARCH-R1
SET P0352 P0006
SFTON P0352
MOVL C00110 BC00110 V=500.0 PL=0
SFTOF
'------------------------
'W250A P
'------------------------
MOVJ C00111 BC00111 VJ=30.00
MOVL C00112 BC00112 V=333.3 PL=0
REFP 3 C00113 BC00113
CALL JOB:SEARCH-R1
IMOV P0058 V=16.7
SET P0353 P0006
SFTON P0353
REFP 3 C00114 BC00114
CALL JOB:SEARCH-R1
SET P0353 P0006
SFTON P0353
MOVL C00115 BC00115 V=500.0 PL=0
SFTOF
'------------------------
'W250A L
'------------------------
MOVJ C00116 BC00116 VJ=30.00
MOVL C00117 BC00117 V=333.3 PL=0
REFP 3 C00118 BC00118
CALL JOB:SEARCH-R1
IMOV P0058 V=16.7
SET P0354 P0006
SFTON P0354
REFP 3 C00119 BC00119
CALL JOB:SEARCH-R1
SET P0354 P0006
SFTON P0354
MOVL C00120 BC00120 V=500.0 PL=0
SFTOF
'------------------------
'W253A P
'------------------------
MOVJ C00121 BC00121 VJ=30.00
MOVL C00122 BC00122 V=333.3 PL=0
REFP 3 C00123 BC00123
CALL JOB:SEARCH-R1
IMOV P0058 V=16.7
SET P0355 P0006
SFTON P0355
REFP 3 C00124 BC00124
CALL JOB:SEARCH-R1
SET P0355 P0006
SFTON P0355
MOVL C00125 BC00125 V=333.3 PL=0
SFTOF
'------------------------
'W253A L
'------------------------
MOVJ C00126 BC00126 VJ=30.00
MOVL C00127 BC00127 V=333.3 PL=0
REFP 3 C00128 BC00128
CALL JOB:SEARCH-R1
IMOV P0058 V=16.7
SET P0356 P0006
SFTON P0356
REFP 3 C00129 BC00129
CALL JOB:SEARCH-R1
SET P0356 P0006
SFTON P0356
MOVL C00130 BC00130 V=500.0 PL=0
SFTOF
'------------------------
'W256A P
'------------------------
MOVJ C00131 BC00131 VJ=30.00
MOVL C00132 BC00132 V=333.3 PL=0
REFP 3 C00133 BC00133
CALL JOB:SEARCH-R1
IMOV P0058 V=16.7
SET P0357 P0006
SFTON P0357
REFP 3 C00134 BC00134
CALL JOB:SEARCH-R1
SET P0357 P0006
SFTON P0357
MOVL C00135 BC00135 V=500.0 PL=0
SFTOF
'------------------------
'W256A L
'------------------------
MOVJ C00136 BC00136 VJ=30.00
MOVL C00137 BC00137 V=333.3 PL=0
REFP 3 C00138 BC00138
CALL JOB:SEARCH-R1
IMOV P0058 V=16.7
SET P0358 P0006
SFTON P0358
REFP 3 C00139 BC00139
CALL JOB:SEARCH-R1
SET P0358 P0006
SFTON P0358
MOVL C00140 BC00140 V=500.0 PL=0
SFTOF
'------------------------
'W252A P
'------------------------
MOVL C00141 BC00141 V=500.0
MOVL C00142 BC00142 V=333.3 PL=0
REFP 3 C00143 BC00143
CALL JOB:SEARCH-R1
IMOV P0058 V=16.7
SET P0359 P0006
SFTON P0359
REFP 3 C00144 BC00144
CALL JOB:SEARCH-R1
SET P0359 P0006
SFTON P0359
MOVL C00145 BC00145 V=333.3 PL=0
SFTOF
'------------------------
'W252A L
'------------------------
MOVL C00146 BC00146 V=500.0
MOVL C00147 BC00147 V=333.3 PL=0
REFP 3 C00148 BC00148
CALL JOB:SEARCH-R1
IMOV P0058 V=16.7
SET P0360 P0006
SFTON P0360
REFP 3 C00149 BC00149
CALL JOB:SEARCH-R1
SET P0360 P0006
SFTON P0360
MOVL C00150 BC00150 V=500.0 PL=0
SFTOF
'------------------------
'W255A
'------------------------
MOVL C00151 BC00151 V=500.0
MOVL C00152 BC00152 V=333.3 PL=0
REFP 3 C00153 BC00153
CALL JOB:SEARCH-R1
IMOV P0058 V=16.7
SET P0361 P0006
SFTON P0361
REFP 3 C00154 BC00154
CALL JOB:SEARCH-R1
SET P0361 P0006
SFTON P0361
MOVL C00155 BC00155 V=500.0 PL=0
SFTOF
MOVL C00156 BC00156 V=500.0
MOVJ C00157 BC00157 VJ=50.00
MOVJ C00158 BC00158 VJ=50.00
MOVJ C00159 BC00159 VJ=50.00
COMM MOVJ C00160 BC00160 VJ=30.00
COMM MOVJ C00161 BC00161 VJ=30.00
COMM MOVJ C00162 BC00162 VJ=30.00
COMM MOVJ C00163 BC00163 VJ=50.00
COMM 'COMMENT
COMM MOVJ C00164 BC00164 VJ=50.00
COMM MOVJ C00165 BC00165 VJ=30.00
COMM GETE D040 P0400 (1)
COMM GETE D041 P0400 (2)
COMM GETE D042 P0400 (3)
COMM SETE P0401 (1) D040
COMM SETE P0401 (2) D041
COMM SETE P0401 (3) D042
COMM GETE D040 P0400 (1)
COMM GETE D041 P0400 (2)
COMM GETE D042 P0400 (3)
COMM SETE P0402 (1) D040
COMM SETE P0402 (2) D041
COMM SETE P0402 (3) D042
COMM MOVL C00166 BC00166 V=333.3
COMM MOVL C00167 BC00167 V=333.3
COMM MOVL C00168 BC00168 V=333.3
COMM MOVL C00169 BC00169 V=333.3
COMM '------------------------
COMM 'W61.5
COMM '------------------------
COMM MOVL C00170 BC00170 V=66.7 PL=0
COMM REFP 3 C00171 BC00171
COMM CALL JOB:SEARCH-R1
COMM SET P0401 P0006
COMM SFTON P0401
COMM MOVL C00172 BC00172 V=66.7 PL=0
COMM REFP 3 C00173 BC00173
COMM CALL JOB:SEARCH-R1
COMM SET P0401 P0006
COMM SFTON P0401
COMM MOVL C00174 BC00174 V=66.7 PL=0
COMM SFTOF
COMM MOVL C00175 BC00175 V=333.3
COMM MOVL C00176 BC00176 V=333.3
COMM '------------------------
COMM 'W61.7
COMM '------------------------
COMM MOVL C00177 BC00177 V=333.3
COMM MOVL C00178 BC00178 V=66.7 PL=0
COMM REFP 3 C00179 BC00179
COMM CALL JOB:SEARCH-R1
COMM SET P0402 P0006
COMM SFTON P0402
COMM MOVL C00180 BC00180 V=66.7 PL=0
COMM REFP 3 C00181 BC00181
COMM CALL JOB:SEARCH-R1
COMM SET P0402 P0006
COMM SFTON P0402
COMM MOVL C00182 BC00182 V=66.7 PL=0
COMM SFTOF
COMM '------------------------
COMM 'W61.10
COMM '------------------------
COMM MOVL C00183 BC00183 V=500.0
COMM MOVL C00184 BC00184 V=166.7 PL=0
COMM REFP 3 C00185 BC00185
COMM CALL JOB:SEARCH-R1
COMM SET P0403 P0006
COMM SFTON P0403
COMM MOVL C00186 BC00186 V=166.7 PL=0
COMM REFP 3 C00187 BC00187
COMM CALL JOB:SEARCH-R1
COMM SET P0403 P0006
COMM SFTON P0403
COMM MOVL C00188 BC00188 V=500.0 PL=0
COMM SFTOF
COMM '------------------------
COMM 'W61.12
COMM '------------------------
COMM MOVL C00189 BC00189 V=500.0
COMM MOVL C00190 BC00190 V=166.7 PL=0
COMM REFP 3 C00191 BC00191
COMM CALL JOB:SEARCH-R1
COMM SET P0404 P0006
COMM SFTON P0404
COMM MOVL C00192 BC00192 V=166.7 PL=0
COMM REFP 3 C00193 BC00193
COMM CALL JOB:SEARCH-R1
COMM SET P0404 P0006
COMM SFTON P0404
COMM MOVL C00194 BC00194 V=500.0 PL=0
COMM SFTOF
COMM '------------------------
COMM 'W61.15
COMM '------------------------
COMM MOVL C00195 BC00195 V=500.0
COMM MOVL C00196 BC00196 V=166.7 PL=0
COMM REFP 3 C00197 BC00197
COMM CALL JOB:SEARCH-R1
COMM SET P0405 P0006
COMM SFTON P0405
COMM MOVL C00198 BC00198 V=166.7 PL=0
COMM REFP 3 C00199 BC00199
COMM CALL JOB:SEARCH-R1
COMM SET P0405 P0006
COMM SFTON P0405
COMM MOVL C00200 BC00200 V=500.0 PL=0
COMM SFTOF
COMM MOVL C00201 BC00201 V=500.0
COMM SFTOF
COMM GETE D040 P0405 (1)
COMM GETE D041 P0405 (2)
COMM GETE D042 P0405 (3)
COMM SETE P0406 (1) D040
COMM SETE P0406 (2) D041
COMM SETE P0406 (3) D042
COMM '------------------------
COMM 'W61.17
COMM '------------------------
COMM MOVL C00202 BC00202 V=333.3
COMM MOVL C00203 BC00203 V=66.7 PL=0
COMM REFP 3 C00204 BC00204
COMM CALL JOB:SEARCH-R1
COMM SET P0406 P0006
COMM SFTON P0406
COMM MOVL C00205 BC00205 V=66.7 PL=0
COMM REFP 3 C00206 BC00206
COMM CALL JOB:SEARCH-R1
COMM SET P0406 P0006
COMM SFTON P0406
COMM MOVL C00207 BC00207 V=66.7 PL=0
COMM SFTOF
COMM MOVL C00208 BC00208 V=333.3
COMM MOVL C00209 BC00209 V=333.3
COMM MOVJ C00210 BC00210 VJ=30.00
COMM MOVJ C00211 BC00211 VJ=50.00
COMM MOVL C00212 BC00212 V=666.7
COMM '------------------------
COMM 'W61.20
COMM '------------------------
COMM MOVL C00213 BC00213 V=500.0
COMM MOVL C00214 BC00214 V=166.7 PL=0
COMM REFP 3 C00215 BC00215
COMM CALL JOB:SEARCH-R1
COMM SET P0407 P0006
COMM SFTON P0407
COMM MOVL C00216 BC00216 V=166.7 PL=0
COMM REFP 3 C00217 BC00217
COMM CALL JOB:SEARCH-R1
COMM SET P0407 P0006
COMM SFTON P0407
COMM MOVL C00218 BC00218 V=500.0 PL=0
COMM SFTOF
COMM '------------------------
COMM 'W61.23
COMM '------------------------
COMM MOVL C00219 BC00219 V=500.0
COMM MOVL C00220 BC00220 V=166.7 PL=0
COMM REFP 3 C00221 BC00221
COMM CALL JOB:SEARCH-R1
COMM SET P0408 P0006
COMM SFTON P0408
COMM MOVL C00222 BC00222 V=166.7 PL=0
COMM REFP 3 C00223 BC00223
COMM CALL JOB:SEARCH-R1
COMM SET P0408 P0006
COMM SFTON P0408
COMM MOVL C00224 BC00224 V=500.0 PL=0
COMM SFTOF
COMM '------------------------
COMM 'W61.25
COMM '------------------------
COMM MOVL C00225 BC00225 V=500.0
COMM MOVL C00226 BC00226 V=166.7 PL=0
COMM REFP 3 C00227 BC00227
COMM CALL JOB:SEARCH-R1
COMM SET P0409 P0006
COMM SFTON P0409
COMM MOVL C00228 BC00228 V=166.7 PL=0
COMM REFP 3 C00229 BC00229
COMM CALL JOB:SEARCH-R1
COMM SET P0409 P0006
COMM SFTON P0409
COMM MOVL C00230 BC00230 V=500.0 PL=0
COMM SFTOF
COMM MOVL C00231 BC00231 V=500.0
COMM MOVL C00232 BC00232 V=500.0
COMM MOVJ C00233 BC00233 VJ=50.00
COMM MOVL C00234 BC00234 V=666.7
COMM GETE D040 P0409 (1)
COMM GETE D041 P0409 (2)
COMM GETE D042 P0409 (3)
COMM SETE P0410 (1) D040
COMM SETE P0410 (2) D041
COMM SETE P0410 (3) D042
COMM '------------------------
COMM 'W61.30
COMM '------------------------
COMM MOVL C00235 BC00235 V=500.0
COMM MOVL C00236 BC00236 V=166.7 PL=0
COMM REFP 3 C00237 BC00237
COMM CALL JOB:SEARCH-R1
COMM SET P0411 P0006
COMM SFTON P0411
COMM MOVL C00238 BC00238 V=166.7 PL=0
COMM REFP 3 C00239 BC00239
COMM CALL JOB:SEARCH-R1
COMM SET P0411 P0006
COMM SFTON P0411
COMM MOVL C00240 BC00240 V=500.0 PL=0
COMM SFTOF
COMM MOVL C00241 BC00241 V=666.7
COMM MOVJ C00242 BC00242 VJ=30.00
MOVJ C00243 BC00243 VJ=50.00
CALL JOB:FRONT_SEARCH_90ST-2_5040
MOVJ C00244 BC00244 VJ=50.00
MOVJ C00245 BC00245 VJ=40.00
MOVJ C00246 BC00246 VJ=30.00
MOVL C00247 BC00247 V=666.7
MOVJ C00248 BC00248 VJ=40.00
'------------------------
'W65.3
'------------------------
SFTON P0300
MOVL C00249 BC00249 V=500.0
MOVL C00250 BC00250 V=333.3 PL=0
MACRO1 MJ#(0) ARGF10
ARCON
MOVL C00251 BC00251 V=10.8
ARCOF
MOVL C00252 BC00252 V=166.7
SFTOF
'------------------------
'W65.5
'------------------------
SFTON P0301
MOVL C00253 BC00253 V=333.3
MOVL C00254 BC00254 V=133.3 PL=0
MACRO1 MJ#(0) ARGF10
ARCON
MOVL C00255 BC00255 V=10.8
ARCOF
MOVL C00256 BC00256 V=166.7
SFTOF
MOVL C00257 BC00257 V=500.0
MOVL C00258 BC00258 V=333.3
MOVJ C00259 BC00259 VJ=25.00
MOVJ C00260 BC00260 VJ=50.00
'::::::::::::::::::::::::::::::::
'::::::::::::::::::::::::::::::::
'::::::::::::::::::::::::::::::::
'::::::::::::::::::::::::::::::::
'::::::::::::::::::::::::::::::::
COMM MOVJ C00261 BC00261 VJ=50.00
COMM MOVJ C00262 BC00262 VJ=50.00
COMM MOVJ C00263 BC00263 VJ=50.00
COMM MOVJ C00264 BC00264 VJ=50.00
COMM MOVJ C00265 BC00265 VJ=20.00
COMM '------------------------
COMM 'W61.3
COMM '------------------------
COMM SFTON P0400
COMM MOVL C00266 BC00266 V=333.3
COMM MOVL C00267 BC00267 V=66.7 PL=0
COMM MACRO1 MJ#(0) ARGF9
COMM ARCOF
COMM SFTOF
COMM 'BELKA PRZEJAZD
COMM MOVJ C00268 BC00268 VJ=25.00
COMM MOVJ C00269 BC00269 VJ=50.00
COMM MOVL C00270 BC00270 V=500.0
COMM MOVL C00271 BC00271 V=500.0
COMM '------------------------
COMM 'W61.5
COMM '------------------------
COMM SFTON P0401
COMM MOVL C00272 BC00272 V=333.3
COMM MOVL C00273 BC00273 V=133.3 PL=0
COMM MACRO1 MJ#(0) ARGF24
COMM ARCON
COMM MOVL C00274 BC00274 V=7.5
COMM ARCOF
COMM MOVL C00275 BC00275 V=250.0
COMM SFTOF
COMM MOVL C00276 BC00276 V=333.3
COMM MOVJ C00277 BC00277 VJ=35.00
COMM MOVJ C00278 BC00278 VJ=50.00
COMM MOVJ C00279 BC00279 VJ=50.00
COMM MOVJ C00280 BC00280 VJ=50.00
MOVJ C00281 BC00281 VJ=50.00
MOVJ C00282 BC00282 VJ=50.00
MOVJ C00283 BC00283 VJ=50.00
'------------------------
'W250A
'------------------------
SFTON P0354
MOVL C00284 BC00284 V=333.3
MOVL C00285 BC00285 V=133.3 PL=0
MACRO1 MJ#(0) ARGF14
ARCON
SFTOF
SFTON P0353
MOVL C00286 BC00286 V=11.7
ARCOF
MOVL C00287 BC00287 V=166.7
SFTOF
MOVJ C00288 BC00288 VJ=50.00
MOVJ C00289 BC00289 VJ=50.00
MOVJ C00290 BC00290 VJ=50.00
MOVJ C00291 BC00291 VJ=50.00
MOVJ C00292 BC00292 VJ=50.00
MOVJ C00293 BC00293 VJ=20.00
MOVJ C00294 BC00294 VJ=10.00
'------------------------
'W65.7
'------------------------
SFTON P0302
'MOTOSIM PULSE LIMIT
MOVL C00295 BC00295 V=500.0
MOVL C00296 BC00296 V=133.3 PL=0
MACRO1 MJ#(0) ARGF10
ARCON
MOVL C00297 BC00297 V=10.8
ARCOF
MOVL C00298 BC00298 V=250.0
SFTOF
'------------------------
'W65.10
'------------------------
SFTON P0303
MOVL C00299 BC00299 V=500.0
MOVL C00300 BC00300 V=166.7 PL=0
ARCON
MOVL C00301 BC00301 V=10.8
ARCOF
MOVL C00302 BC00302 V=166.7
SFTOF
SFTOF
MOVL C00303 BC00303 V=333.3
MOVL C00304 BC00304 V=500.0
MOVJ C00305 BC00305 VJ=50.00
MOVJ C00306 BC00306 VJ=30.00
MOVJ C00307 BC00307 VJ=50.00
MOVJ C00308 BC00308 VJ=50.00
COMM '::::::::::::::::::::::::::::::::
COMM '::::::::::::::::::::::::::::::::
COMM '------------------------
COMM 'W61.7
COMM '------------------------
COMM '::::::::::::::::::::::::::::::::
COMM '::::::::::::::::::::::::::::::::
COMM MOVJ C00309 BC00309 VJ=50.00
COMM MOVJ C00310 BC00310 VJ=35.00
COMM SFTON P0402
COMM MOVL C00311 BC00311 V=333.3
COMM MOVL C00312 BC00312 V=133.3 PL=0
COMM MACRO1 MJ#(0) ARGF24
COMM ARCON
COMM MOVL C00313 BC00313 V=7.5
COMM ARCOF
COMM MOVL C00314 BC00314 V=166.7
COMM SFTOF
COMM MOVL C00315 BC00315 V=500.0
COMM MOVL C00316 BC00316 V=500.0
COMM MOVJ C00317 BC00317 VJ=50.00
COMM '------------------------
COMM 'W61.10
COMM '------------------------
COMM SFTON P0403
COMM MOVL C00318 BC00318 V=333.3
COMM MOVL C00319 BC00319 V=133.3 PL=0
COMM MACRO1 MJ#(0) ARGF24
COMM ARCON
COMM MOVL C00320 BC00320 V=7.5
COMM ARCOF
COMM MOVL C00321 BC00321 V=166.7
COMM SFTOF
COMM MOVL C00322 BC00322 V=333.3
COMM MOVJ C00323 BC00323 VJ=35.00
COMM MOVJ C00324 BC00324 VJ=50.00
COMM MOVJ C00325 BC00325 VJ=50.00
COMM '::::::::::::::::::::::::
COMM '::::::::::::::::::::::::
COMM '::::::::::::::::::::::::
COMM '::::::::::::::::::::::::
COMM '::::::::::::::::::::::::
COMM '::::::::::::::::::::::::
COMM '::::::::::::::::::::::::
MOVJ C00326 BC00326 VJ=50.00
MOVJ C00327 BC00327 VJ=50.00
MOVJ C00328 BC00328 VJ=50.00
'------------------------
'W214A
'------------------------
SFTON P0350
MOVL C00329 BC00329 V=333.3
MOVL C00330 BC00330 V=333.3
MOVL C00331 BC00331 V=133.3 PL=0
MACRO1 MJ#(0) ARGF14
ARCON
SFTOF
SFTON P0350
MOVL C00332 BC00332 V=11.7
ARCOF
MOVL C00333 BC00333 V=250.0
SFTOF
MOVJ C00334 BC00334 VJ=50.00
MOVJ C00335 BC00335 VJ=50.00
MOVJ C00336 BC00336 VJ=50.00
MOVJ C00337 BC00337 VJ=50.00
MOVJ C00338 BC00338 VJ=50.00
MOVJ C00339 BC00339 VJ=50.00
MOVJ C00340 BC00340 VJ=20.00
'------------------------
'W65.12
'------------------------
SFTON P0304
MOVL C00341 BC00341 V=333.3
MOVL C00342 BC00342 V=133.3 PL=0
MACRO1 MJ#(0) ARGF10
ARCON
MOVL C00343 BC00343 V=10.8
ARCOF
MOVL C00344 BC00344 V=166.7
SFTOF
'------------------------
'W65.15
'------------------------
SFTON P0305
MOVL C00345 BC00345 V=333.3
MOVL C00346 BC00346 V=166.7 PL=0
MACRO1 MJ#(0) ARGF10
ARCON
MOVL C00347 BC00347 V=10.8
ARCOF
MOVL C00348 BC00348 V=166.7
SFTOF
MOVL C00349 BC00349 V=333.3
MOVL C00350 BC00350 V=500.0
MOVL C00351 BC00351 V=500.0
MOVJ C00352 BC00352 VJ=50.00
COMM '::::::::::::::::::::::::
COMM '::::::::::::::::::::::::
COMM '::::::::::::::::::::::::
COMM '::::::::::::::::::::::::
COMM '::::::::::::::::::::::::
COMM '::::::::::::::::::::::::
COMM '::::::::::::::::::::::::
COMM MOVJ C00353 BC00353 VJ=50.00
COMM MOVJ C00354 BC00354 VJ=50.00
COMM '::::::::::::::::::::::::::::::::
COMM '::::::::::::::::::::::::::::::::
COMM '------------------------
COMM 'W61.12
COMM '------------------------
COMM '::::::::::::::::::::::::::::::::
COMM '::::::::::::::::::::::::::::::::
COMM SFTON P0404
COMM MOVJ C00355 BC00355 VJ=50.00
COMM MOVL C00356 BC00356 V=333.3
COMM MOVL C00357 BC00357 V=333.3
COMM MOVL C00358 BC00358 V=166.7 PL=0
COMM MACRO1 MJ#(0) ARGF24
COMM ARCON
COMM MOVL C00359 BC00359 V=7.5
COMM ARCOF
COMM MOVL C00360 BC00360 V=166.7
COMM SFTOF
COMM MOVL C00361 BC00361 V=333.3
COMM MOVL C00362 BC00362 V=333.3
COMM '------------------------
COMM 'W61.15
COMM '------------------------
COMM SFTON P0405
COMM MOVL C00363 BC00363 V=333.3
COMM MOVL C00364 BC00364 V=166.7 PL=0
COMM MACRO1 MJ#(0) ARGF24
COMM ARCON
COMM MOVL C00365 BC00365 V=7.5
COMM ARCOF
COMM MOVL C00366 BC00366 V=166.7
COMM SFTOF
COMM MOVJ C00367 BC00367 VJ=50.00
COMM MOVJ C00368 BC00368 VJ=50.00
COMM MOVJ C00369 BC00369 VJ=50.00
COMM '::::::::::::::::::::::::
COMM '::::::::::::::::::::::::
COMM '::::::::::::::::::::::::
COMM '::::::::::::::::::::::::
COMM '::::::::::::::::::::::::
COMM '::::::::::::::::::::::::
COMM '::::::::::::::::::::::::
MOVJ C00370 BC00370 VJ=50.00
MOVJ C00371 BC00371 VJ=50.00
'------------------------
'W252A
'------------------------
SFTON P0359
MOVL C00372 BC00372 V=500.0
MOVL C00373 BC00373 V=166.7 PL=0
MACRO1 MJ#(0) ARGF14
ARCON
SFTOF
SFTON P0358
MOVL C00374 BC00374 V=11.7
ARCOF
MOVL C00375 BC00375 V=250.0
SFTOF
MOVJ C00376 BC00376 VJ=50.00
MOVJ C00377 BC00377 VJ=80.00
MOVJ C00378 BC00378 VJ=80.00
MOVJ C00379 BC00379 VJ=50.00
MOVJ C00380 BC00380 VJ=50.00
MOVJ C00381 BC00381 VJ=25.00
MOVL C00382 BC00382 V=333.3
MOVL C00383 BC00383 V=333.3
'------------------------
'W65.17
'------------------------
SFTON P0306
MOVL C00384 BC00384 V=166.7
MOVL C00385 BC00385 V=166.7 PL=0
MACRO1 MJ#(0) ARGF10
ARCON
MOVL C00386 BC00386 V=10.8
ARCOF
MOVL C00387 BC00387 V=166.7
SFTOF
MOVL C00388 BC00388 V=250.0
MOVL C00389 BC00389 V=250.0
MOVL C00390 BC00390 V=333.3
MOVJ C00391 BC00391 VJ=25.00
'::::::::::::::::::::::::
'::::::::::::::::::::::::
'::::::::::::::::::::::::
'::::::::::::::::::::::::
'::::::::::::::::::::::::
'::::::::::::::::::::::::
'::::::::::::::::::::::::
'::::::::::::::::::::::::::::::::
'::::::::::::::::::::::::::::::::
'------------------------
'W61.17
'------------------------
'::::::::::::::::::::::::::::::::
'::::::::::::::::::::::::::::::::
COMM SFTON P0406
COMM MOVJ C00392 BC00392 VJ=10.00
COMM MOVL C00393 BC00393 V=150.0
COMM MOVL C00394 BC00394 V=66.7 PL=0
COMM MACRO1 MJ#(0) ARGF24
COMM ARCON
COMM MOVL C00395 BC00395 V=6.7
COMM ARCOF
COMM MOVL C00396 BC00396 V=83.3
COMM SFTOF
'------------------------
'W253A
'------------------------
MOVJ C00397 BC00397 VJ=50.00
MOVJ C00398 BC00398 VJ=50.00
SFTON P0356
MOVL C00399 BC00399 V=333.3
MOVL C00400 BC00400 V=333.3
MOVL C00401 BC00401 V=166.7 PL=0
MACRO1 MJ#(0) ARGF14
ARCON
SFTOF
SFTON P0355
MOVL C00402 BC00402 V=11.7
ARCOF
MOVL C00403 BC00403 V=250.0
SFTOF
MOVJ C00404 BC00404 VJ=50.00
MOVJ C00405 BC00405 VJ=50.00
MOVJ C00406 BC00406 VJ=80.00
MOVJ C00407 BC00407 VJ=80.00
MOVJ C00408 BC00408 VJ=50.00
MOVJ C00409 BC00409 VJ=50.00
MOVJ C00410 BC00410 VJ=50.00
MOVJ C00411 BC00411 VJ=30.00
MOVJ C00412 BC00412 VJ=30.00
'------------------------
'W65.20
'------------------------
SFTON P0307
MOVL C00413 BC00413 V=333.3
MOVL C00414 BC00414 V=166.7
MOVL C00415 BC00415 V=166.7 PL=0
MACRO1 MJ#(0) ARGF10
ARCON
MOVL C00416 BC00416 V=10.8
ARCOF
MOVL C00417 BC00417 V=250.0
SFTOF
MOVL C00418 BC00418 V=333.3
MOVL C00419 BC00419 V=333.3
MOVL C00420 BC00420 V=333.3
MOVJ C00421 BC00421 VJ=50.00
MOVJ C00422 BC00422 VJ=50.00
MOVJ C00423 BC00423 VJ=50.00
MOVJ C00424 BC00424 VJ=50.00
COMM '::::::::::::::::::::::::
COMM '::::::::::::::::::::::::
COMM '::::::::::::::::::::::::
COMM '::::::::::::::::::::::::
COMM '::::::::::::::::::::::::
COMM '::::::::::::::::::::::::
COMM '::::::::::::::::::::::::
COMM MOVJ C00425 BC00425 VJ=80.00
COMM MOVJ C00426 BC00426 VJ=50.00
COMM MOVJ C00427 BC00427 VJ=50.00
COMM '::::::::::::::::::::::::::::::::
COMM '::::::::::::::::::::::::::::::::
COMM '------------------------
COMM 'W61.20
COMM '------------------------
COMM '::::::::::::::::::::::::::::::::
COMM '::::::::::::::::::::::::::::::::
COMM SFTON P0407
COMM MOVL C00428 BC00428 V=333.3
COMM MOVL C00429 BC00429 V=166.7
COMM MOVL C00430 BC00430 V=133.3 PL=0
COMM MACRO1 MJ#(0) ARGF24
COMM ARCON
COMM MOVL C00431 BC00431 V=7.5
COMM ARCOF
COMM MOVL C00432 BC00432 V=166.7
COMM SFTOF
COMM SFTON P0407
COMM MOVL C00433 BC00433 V=166.7
COMM MOVL C00434 BC00434 V=133.3 PL=0
COMM MACRO1 MJ#(0) ARGF24
COMM ARCON
COMM MOVL C00435 BC00435 V=7.5
COMM ARCOF
COMM MOVL C00436 BC00436 V=166.7
COMM SFTOF
COMM '::::::::::::::::::::::::
COMM '::::::::::::::::::::::::
COMM '::::::::::::::::::::::::
COMM '::::::::::::::::::::::::
COMM '::::::::::::::::::::::::
COMM MOVJ C00437 BC00437 VJ=50.00
COMM MOVJ C00438 BC00438 VJ=50.00
COMM MOVJ C00439 BC00439 VJ=50.00
COMM MOVJ C00440 BC00440 VJ=50.00
COMM '------------------------
COMM 'W254A
COMM '------------------------
MOVJ C00441 BC00441 VJ=50.00
MOVJ C00442 BC00442 VJ=50.00
SFTON P0352
MOVL C00443 BC00443 V=500.0
MOVL C00444 BC00444 V=500.0
MOVL C00445 BC00445 V=166.7 PL=0
MACRO1 MJ#(0) ARGF14
ARCON
SFTOF
SFTON P0351
MOVL C00446 BC00446 V=11.7
ARCOF
MOVL C00447 BC00447 V=333.3
SFTOF
COMM MOVJ C00448 BC00448 VJ=80.00
COMM MOVJ C00449 BC00449 VJ=80.00
COMM MOVJ C00450 BC00450 VJ=80.00
COMM MOVJ C00451 BC00451 VJ=80.00
COMM MOVJ C00452 BC00452 VJ=50.00
MOVJ C00453 BC00453 VJ=50.00
MOVJ C00454 BC00454 VJ=50.00
MOVJ C00455 BC00455 VJ=50.00
MOVJ C00456 BC00456 VJ=30.00
MOVL C00457 BC00457 V=500.0
'------------------------
'W65.23
'------------------------
SFTON P0308
MOVL C00458 BC00458 V=333.3
MOVL C00459 BC00459 V=166.7
MOVL C00460 BC00460 V=133.3 PL=0
MACRO1 MJ#(0) ARGF10
ARCON
MOVL C00461 BC00461 V=10.8
ARCOF
MOVL C00462 BC00462 V=166.7
SFTOF
'------------------------
'W65.25
'------------------------
SFTON P0309
MOVL C00463 BC00463 V=500.0
MOVL C00464 BC00464 V=133.3 PL=0
ARCON
MOVL C00465 BC00465 V=10.8
ARCOF
MOVL C00466 BC00466 V=166.7
SFTOF
MOVL C00467 BC00467 V=500.0
MOVL C00468 BC00468 V=333.3
MOVL C00469 BC00469 V=500.0
MOVL C00470 BC00470 V=333.3
MOVJ C00471 BC00471 VJ=50.00
MOVJ C00472 BC00472 VJ=50.00
MOVJ C00473 BC00473 VJ=50.00
MOVJ C00474 BC00474 VJ=80.00
COMM '::::::::::::::::::::::::
COMM '::::::::::::::::::::::::
COMM '::::::::::::::::::::::::
COMM '::::::::::::::::::::::::
COMM '::::::::::::::::::::::::
COMM '::::::::::::::::::::::::
COMM '::::::::::::::::::::::::
COMM MOVJ C00475 BC00475 VJ=80.00
COMM MOVJ C00476 BC00476 VJ=80.00
COMM MOVJ C00477 BC00477 VJ=50.00
COMM MOVJ C00478 BC00478 VJ=50.00
COMM '::::::::::::::::::::::::::::::::
COMM '::::::::::::::::::::::::::::::::
COMM '------------------------
COMM 'W61.23
COMM '------------------------
COMM '::::::::::::::::::::::::::::::::
COMM '::::::::::::::::::::::::::::::::
COMM SFTON P0408
COMM MOVL C00479 BC00479 V=333.3
COMM MOVL C00480 BC00480 V=166.7
COMM MOVL C00481 BC00481 V=133.3 PL=0
COMM MACRO1 MJ#(0) ARGF24
COMM ARCON
COMM MOVL C00482 BC00482 V=7.5
COMM ARCOF
COMM MOVL C00483 BC00483 V=83.3
COMM SFTOF
COMM '------------------------
COMM 'W61.25
COMM '------------------------
COMM SFTON P0409
COMM MOVL C00484 BC00484 V=333.3
COMM MOVL C00485 BC00485 V=150.0
COMM MOVL C00486 BC00486 V=133.3 PL=0
COMM MACRO1 MJ#(0) ARGF24
COMM ARCON
COMM MOVL C00487 BC00487 V=7.5
COMM ARCOF
COMM MOVL C00488 BC00488 V=166.7
COMM SFTOF
COMM '::::::::::::::::::::::::
COMM '::::::::::::::::::::::::
COMM '::::::::::::::::::::::::
COMM '::::::::::::::::::::::::
COMM '::::::::::::::::::::::::
COMM MOVL C00489 BC00489 V=333.3
COMM MOVJ C00490 BC00490 VJ=50.00
COMM MOVJ C00491 BC00491 VJ=50.00
COMM MOVJ C00492 BC00492 VJ=50.00
COMM MOVJ C00493 BC00493 VJ=50.00
MOVJ C00494 BC00494 VJ=80.00
'------------------------
'W255A
MOVL C00495 BC00495 V=500.0
MOVL C00496 BC00496 V=333.3
SFTON P0361
MOVL C00497 BC00497 V=133.3 PL=0
MACRO1 MJ#(0) ARGF14
ARCON
MOVL C00498 BC00498 V=11.7
ARCOF
MOVL C00499 BC00499 V=250.0
SFTOF
MOVL C00500 BC00500 V=333.3
MOVL C00501 BC00501 V=333.3
MOVL C00502 BC00502 V=500.0
MOVJ C00503 BC00503 VJ=50.00
MOVJ C00504 BC00504 VJ=50.00
MOVJ C00505 BC00505 VJ=80.00
MOVJ C00506 BC00506 VJ=50.00
MOVJ C00507 BC00507 VJ=50.00
MOVL C00508 BC00508 V=333.3
'------------------------
'W31.28
'------------------------
SFTON P0310
MOVL C00509 BC00509 V=333.3
MOVL C00510 BC00510 V=333.3
MOVL C00511 BC00511 V=166.7
COMM MOVL C00512 BC00512 V=66.7 PL=0
COMM MACRO1 MJ#(0) ARGF24
COMM ARCON
COMM MOVL C00513 BC00513 V=8.3
COMM ARCOF
MOVL C00514 BC00514 V=83.3
SFTOF
'------------------------
'W31.30
'------------------------
SFTON P0311
MOVL C00515 BC00515 V=333.3
MOVL C00516 BC00516 V=133.3 PL=0
MACRO1 MJ#(0) ARGF10
ARCON
MOVL C00517 BC00517 V=10.8
ARCOF
MOVL C00518 BC00518 V=166.7
SFTOF
MOVL C00519 BC00519 V=333.3
MOVL C00520 BC00520 V=500.0
MOVL C00521 BC00521 V=333.3
'::::::::::::::::::::::::
'::::::::::::::::::::::::
'::::::::::::::::::::::::
'::::::::::::::::::::::::
'::::::::::::::::::::::::
'::::::::::::::::::::::::
'::::::::::::::::::::::::
MOVJ C00522 BC00522 VJ=50.00 PL=0
COMM MOVJ C00523 BC00523 VJ=50.00
COMM MOVJ C00524 BC00524 VJ=50.00
COMM '::::::::::::::::::::::::::::::::
COMM '::::::::::::::::::::::::::::::::
COMM '------------------------
COMM 'W61.30
COMM '------------------------
COMM '::::::::::::::::::::::::::::::::
COMM '::::::::::::::::::::::::::::::::
COMM SFTON P0411
COMM MOVL C00525 BC00525 V=333.3
COMM MOVL C00526 BC00526 V=133.3 PL=0
COMM MACRO1 MJ#(0) ARGF24
COMM ARCON
COMM MOVL C00527 BC00527 V=7.5
COMM ARCOF
COMM MOVL C00528 BC00528 V=166.7
COMM SFTOF
COMM MOVL C00529 BC00529 V=500.0
COMM MOVJ C00530 BC00530 VJ=50.00
COMM MOVJ C00531 BC00531 VJ=50.00
COMM MOVJ C00532 BC00532 VJ=50.00
COMM MOVJ C00533 BC00533 VJ=80.00
COMM MOVJ C00534 BC00534 VJ=80.00
COMM '------------------------
COMM 'W256A
COMM '------------------------
MOVJ C00535 BC00535 VJ=80.00
MOVJ C00536 BC00536 VJ=80.00
SFTON P0358
MOVL C00537 BC00537 V=333.3
MOVL C00538 BC00538 V=250.0
MOVL C00539 BC00539 V=166.7 PL=0
MACRO1 MJ#(0) ARGF14
ARCON
SFTOF
SFTON P0357
MOVL C00540 BC00540 V=11.7
ARCOF
MOVL C00541 BC00541 V=333.3
SFTOF
MOVJ C00542 BC00542 VJ=50.00
MOVJ C00543 BC00543 VJ=50.00
MOVJ C00544 BC00544 VJ=80.00
CALL JOB:FRONT_WELD_90ST-2_5040
CALL JOB:MOVE_OUT_OF_TUNNEL
END
